TYPE ST_SettingsAX5000 :
STRUCT
	{warning '#TODO: ADD setting during development'}
	rMaxTargetSpeed : LREAL := 200.0; /// Maximum target speed [default: 200.0 mm/s]
END_STRUCT
END_TYPE

(* stored: Version 1.1.0.1, ProductVersion 3.1.4024.12
   DUT ST_SettingsAX5000: Id {ed6a1034-fbc2-4d8e-a32e-f51a7b4f2923} *)
